PROGRAM Axis04_Auto
VAR
//System_Bit
	Always_ON	:	BOOL	:=TRUE	;//상시 ON 
	Always_OFF	:	BOOL	:=FALSE	;//상시 OFF
END_VAR
VAR // added by the converter: edge detectors and wires of the graphical bodies
    _rt1 : R_TRIG;
END_VAR

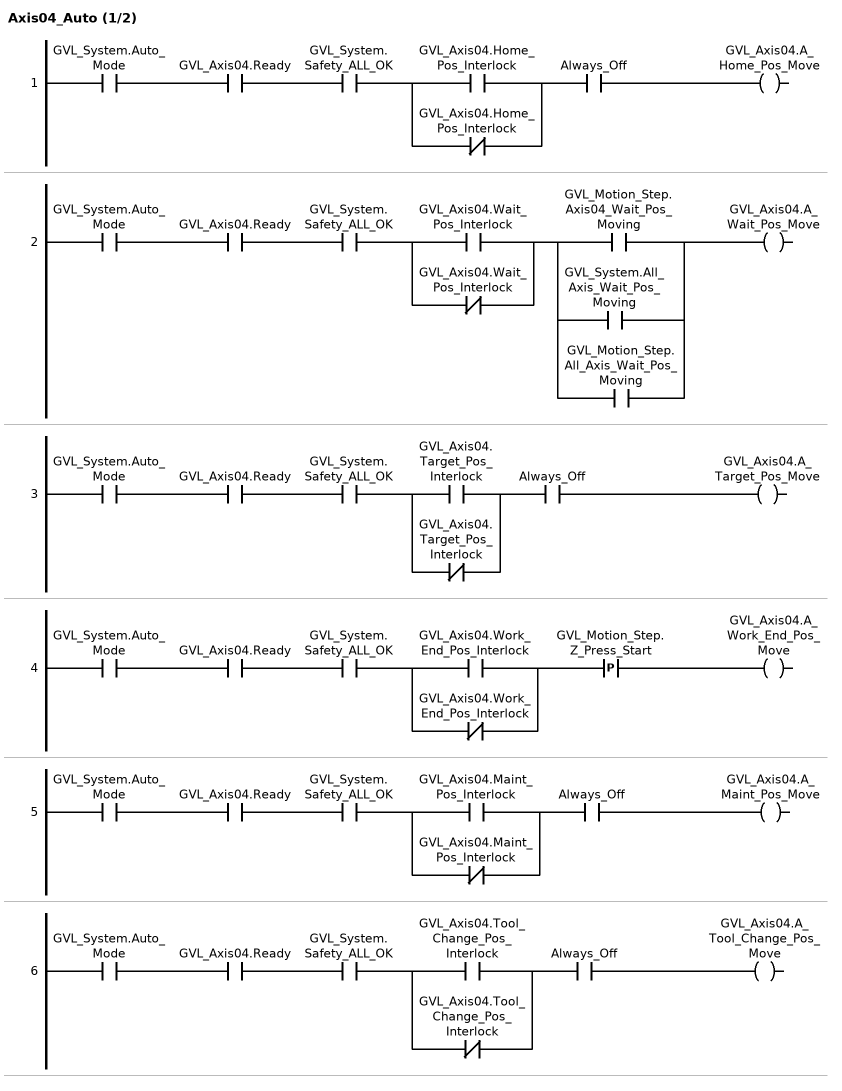
// NETWORK 1
GVL_Axis04.A_Home_Pos_Move := GVL_System.Auto_Mode AND GVL_Axis04.Ready AND GVL_System.Safety_ALL_OK AND (GVL_Axis04.Home_Pos_Interlock OR NOT GVL_Axis04.Home_Pos_Interlock) AND Always_Off;

// NETWORK 2
GVL_Axis04.A_Wait_Pos_Move := GVL_System.Auto_Mode AND GVL_Axis04.Ready AND GVL_System.Safety_ALL_OK AND (GVL_Axis04.Wait_Pos_Interlock OR NOT GVL_Axis04.Wait_Pos_Interlock) AND (GVL_Motion_Step.Axis04_Wait_Pos_Moving OR GVL_System.All_Axis_Wait_Pos_Moving OR GVL_Motion_Step.All_Axis_Wait_Pos_Moving);

// NETWORK 3
GVL_Axis04.A_Target_Pos_Move := GVL_System.Auto_Mode AND GVL_Axis04.Ready AND GVL_System.Safety_ALL_OK AND (GVL_Axis04.Target_Pos_Interlock OR NOT GVL_Axis04.Target_Pos_Interlock) AND Always_Off;

// NETWORK 4
_rt1(CLK := GVL_Motion_Step.Z_Press_Start);
GVL_Axis04.A_Work_End_Pos_Move := GVL_System.Auto_Mode AND GVL_Axis04.Ready AND GVL_System.Safety_ALL_OK AND (GVL_Axis04.Work_End_Pos_Interlock OR NOT GVL_Axis04.Work_End_Pos_Interlock) AND _rt1.Q;

// NETWORK 5
GVL_Axis04.A_Maint_Pos_Move := GVL_System.Auto_Mode AND GVL_Axis04.Ready AND GVL_System.Safety_ALL_OK AND (GVL_Axis04.Maint_Pos_Interlock OR NOT GVL_Axis04.Maint_Pos_Interlock) AND Always_Off;

// NETWORK 6
GVL_Axis04.A_Tool_Change_Pos_Move := GVL_System.Auto_Mode AND GVL_Axis04.Ready AND GVL_System.Safety_ALL_OK AND (GVL_Axis04.Tool_Change_Pos_Interlock OR NOT GVL_Axis04.Tool_Change_Pos_Interlock) AND Always_Off;

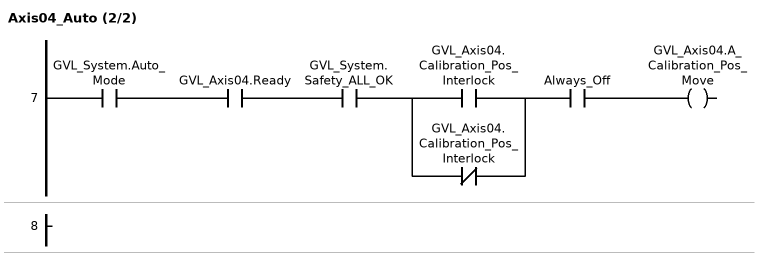
// NETWORK 7
GVL_Axis04.A_Calibration_Pos_Move := GVL_System.Auto_Mode AND GVL_Axis04.Ready AND GVL_System.Safety_ALL_OK AND (GVL_Axis04.Calibration_Pos_Interlock OR NOT GVL_Axis04.Calibration_Pos_Interlock) AND Always_Off;

// NETWORK 8

END_PROGRAM

(* stored: Version 1.1.0.1, ProductVersion 3.1.4024.15
   POU Axis04_Auto: Id {0735a1ba-c4fd-4580-8e71-47f2213f5fd9}, SpecialFunc None *)
